{attribute 'GeneratedUsingTerminal: AT2050-0501-0021'}
{attribute addProperty BoxType "AT2050-0501-0021"}
{attribute addProperty Id "A_0086_AT2050_5500_0019_AT2050_5500AT2050_33A3DF1B80"}
{attribute addProperty CRC "3717075088"}
{attribute addProperty Size "80"}
TYPE A_0058_AT2050_0501_0021_DD8E1090 EXTENDS AT2050_2EA6C9BF :
STRUCT
	{attribute addProperty Name "A_0086_AT2050_5500_0019_AT2050_5500"}
	{attribute addProperty PreviousPort "A_0058(AT2050-0501-0021) : B"}
	A_0086_AT2050_5500_0019_AT2050_5500 : AT2050_33A3DF1B;
END_STRUCT
END_TYPE

(* stored: Version 1.2.0.0, ProductVersion 3.1.4024.9
   DUT A_0058_AT2050_0501_0021_DD8E1090: Id {e162b216-d626-48b8-a890-ce9fc97cdf24} *)
